// TwinCAT 3 PLC project WashingMachineSimulator
// ProgramVersion: 3.1.4024.0
// libraries:
//   Tc2_Standard, * (Beckhoff Automation GmbH)
//   Tc2_System, * (Beckhoff Automation GmbH)
//   Tc3_Module, * (Beckhoff Automation GmbH)
// project tree:
//   / Class Diagram.TcCD (not stored), PlcTask.TcTTO
//   DUTs/ E_MachineState.TcDUT, E_Strategy.TcDUT, ST_Wash.TcDUT
//   GVLs/ GVL_References.TcGVL
//   POUs/ Class Diagram_1.TcCD (not stored), Class Diagram_2.TcCD (not stored), FB_WashingMachine.TcPOU, MAIN.TcPOU
//   POUs/Motor/ FB_BaseMotor.TcPOU, I_Motor.TcIO
//   POUs/Pump/ FB_WaterController.TcPOU, I_WaterController.TcIO
//   POUs/Strategies/ FB_HeavyWash.TcPOU, FB_NormalWash.TcPOU, FB_SoftWash.TcPOU, I_WashStrategy.TcIO
// real-time tasks:
//   TASK PlcTask: cycle T#10ms, priority 20, ADS port 350

CONFIGURATION WashingMachineSimulator
    RESOURCE PLC ON TwinCAT3
        TASK PlcTask(INTERVAL := T#10ms, PRIORITY := 20);
        PROGRAM MAIN WITH PlcTask : MAIN;
    END_RESOURCE
END_CONFIGURATION

// ---- DUTs/E_MachineState.TcDUT
{attribute 'qualified_only'}
{attribute 'strict'}
TYPE E_MachineState :
(
	IDLE := 0,
	CONFIGURING,
	FILLING,
	WASHING,
	DRAINING,
	COMPLETED,
	DRYING,
	ERROR
);
END_TYPE

// ---- DUTs/E_Strategy.TcDUT
{attribute 'qualified_only'}
{attribute 'strict'}
TYPE E_Strategy :
(
	SOFT := 0,
	NORMAL,
	HEAVY
);
END_TYPE

// ---- DUTs/ST_Wash.TcDUT
TYPE ST_Wash :
STRUCT
	nWaterLevel : INT := 1 ;
	eWashStrategy : E_Strategy := E_Strategy.SOFT;
	
END_STRUCT
END_TYPE

// ---- GVLs/GVL_References.TcGVL
{attribute 'qualified_only'}
VAR_GLOBAL
	fbSoftWash : FB_SoftWash;
	fbNormalWash : FB_NormalWash;
	fbHeavyWash : FB_HeavyWash;
	
	fbMotor : FB_BaseMotor;
	fbWaterController : FB_WaterController;
END_VAR

// ---- POUs/Motor/I_Motor.TcIO
INTERFACE I_Motor

METHOD DrySpin 
VAR_INPUT
	nMotorSpeed : INT;
END_VAR
END_METHOD

METHOD Stop
VAR_INPUT
END_VAR
END_METHOD

METHOD WashSpin 
VAR_INPUT
	nMotorSpeed : INT;
END_VAR
END_METHOD

END_INTERFACE

// ---- POUs/Pump/I_WaterController.TcIO
INTERFACE I_WaterController

METHOD GetDuration : TIME
VAR_INPUT
	stWash : REFERENCE TO ST_Wash;
END_VAR
END_METHOD

METHOD StartDrain : BOOL
VAR_INPUT
END_VAR
END_METHOD

METHOD StartFill : BOOL
VAR_INPUT
END_VAR
END_METHOD

METHOD Stop
END_METHOD

END_INTERFACE

// ---- POUs/Strategies/I_WashStrategy.TcIO
INTERFACE I_WashStrategy

METHOD GetDuration : TIME
END_METHOD

METHOD GetRinseCount : INT
END_METHOD

METHOD StartSpin : BOOL
END_METHOD

METHOD StartWash : BOOL
VAR_INPUT
	iMotor : I_Motor;
END_VAR
END_METHOD

METHOD Stop
END_METHOD

END_INTERFACE

// ---- POUs/MAIN.TcPOU
PROGRAM MAIN
VAR
	stWash1 : ST_Wash := (nWaterLevel := 4, eWashStrategy := E_Strategy.NORMAL );
	
	fbWashingMachine : FB_WashingMachine();
	bStart: BOOL;
	
	eWashingMachineState : E_MachineState;
	tRemainingTime : TIME;
END_VAR

IF bStart THEN
	fbWashingMachine.Start();
END_IF
fbWashingMachine(stWash := stWash1);
eWashingMachineState := fbWashingMachine.eState;
tRemainingTime := fbWashingMachine.tRemainingTime;

END_PROGRAM

// ---- POUs/FB_WashingMachine.TcPOU
FUNCTION_BLOCK FB_WashingMachine

VAR_IN_OUT
	stWash : ST_Wash;
END_VAR
VAR
	iWashStrategy : I_WashStrategy;
	iMotor : I_Motor;
	iWaterController : I_WaterController;
	
	eMachineState : E_MachineState;
	tTotalTime : TIME ;
	bRunning : BOOL;
	tBaseTime : TIME := T#5S;
	tRemainingWashingTime : TIME ;
	nRinseCount : INT;
	
	fbTimer : TON ;
END_VAR


IF tTotalTime <> T#0S THEN
	fbTimer (IN := bRunning , PT := tTotalTime);
	tRemainingTime := fbTimer.PT - fbTimer.ET;
END_IF

IF __ISVALIDREF(stWash) THEN
	
	CASE eMachineState OF
		E_MachineState.IDLE:
			IF bRunning THEN
				eMachineState := E_MachineState.CONFIGURING;
			END_IF
			
		E_MachineState.CONFIGURING:
			nRinseCount := 0;
			iWashStrategy := SelectStrategy();
			iMotor := SelectMotor();
			iWaterController := SelectWaterController();
			IF iWashStrategy <> 0 AND iWaterController <> 0 AND iMotor <> 0 THEN
				tTotalTime := iWaterController.GetDuration(stWash) * iWashStrategy.GetRinseCount() + iWashStrategy.GetDuration();
				tRemainingTime := tTotalTime;
				eMachineState := E_MachineState.FILLING;
			ELSE
				eMachineState := E_MachineState.ERROR;
			END_IF
		
		E_MachineState.FILLING:
			IF NOT iWaterController.StartFill() THEN
				eMachineState := E_MachineState.WASHING;
			END_IF
				
		E_MachineState.WASHING:
			IF iWashStrategy.StartWash(iMotor) THEN
				eMachineState := E_MachineState.DRAINING;
			END_IF
		
		E_MachineState.DRAINING:
				IF NOT iWaterController.StartDrain() THEN
					nRinseCount := nRinseCount + 1;
					IF nRinseCount = iWashStrategy.GetRinseCount() THEN
						eMachineState := E_MachineState.DRYING;
					ELSE
						eMachineState := E_MachineState.FILLING;
					END_IF
				END_IF
				
		E_MachineState.DRYING:
			IF iWashStrategy.StartSpin() THEN
				eMachineState := E_MachineState.COMPLETED;
			END_IF
			
		E_MachineState.COMPLETED:
			Stop();
			fbTimer( IN := bRunning);
			tTotalTime := T#0S;
			tRemainingTime := tTotalTime;
			
		E_MachineState.ERROR:
			Stop();
			
		
	END_CASE
	
END_IF

PROPERTY eState : E_MachineState
GET
eState := eMachineState;
END_GET
SET // PRIVATE
eMachineState := eState;
END_SET
END_PROPERTY

METHOD PRIVATE SelectMotor : I_Motor
SelectMotor := GVL_References.fbMotor;
END_METHOD

METHOD PRIVATE SelectStrategy : I_WashStrategy
CASE stWash.eWashStrategy OF
	E_Strategy.SOFT :
	SelectStrategy :=  GVL_References.fbSoftWash;
	
	E_Strategy.NORMAL :
	SelectStrategy :=  GVL_References.fbNormalWash;
	
	E_Strategy.HEAVY :
	SelectStrategy :=  GVL_References.fbHeavyWash;
	
END_CASE
END_METHOD

METHOD PRIVATE SelectWaterController : I_WaterController
SelectWaterController :=  GVL_References.fbWaterController;
END_METHOD

METHOD Start
bRunning := TRUE;
END_METHOD

METHOD Stop
bRunning := FALSE;
END_METHOD

PROPERTY tRemainingTime : TIME
GET
tRemainingTime := tRemainingWashingTime;
END_GET
SET // PRIVATE
tRemainingWashingTime := tRemainingTime;
END_SET
END_PROPERTY

END_FUNCTION_BLOCK

// ---- POUs/Strategies/FB_SoftWash.TcPOU
FUNCTION_BLOCK FB_SoftWash IMPLEMENTS I_WashStrategy

VAR
	nWashCount : INT := 1;
	nRinseCount : INT := 1;
	iMotorRef : I_Motor;
	bWashing : BOOL;
	bDrying : BOOL;
	
	tWashTime : TIME := T#10S;
	nMotorWashSpeed : INT := 100;
	
	nMotorDrySpeed : INT := 700; 
	nMotorDryTime : TIME := T#7S;
	
	fbWashTimer : TON;
END_VAR

{warning 'add method implementation '}
METHOD GetDuration : TIME
VAR
END_VAR
GetDuration := tWashTime * (nRinseCount + nWashCount) + nMotorDryTime ;
END_METHOD

METHOD GetRinseCount : INT
VAR_INPUT
END_VAR
GetRinseCount := nRinseCount + nWashCount;
END_METHOD

METHOD StartSpin : BOOL
bDrying := TRUE;
fbWashTimer( IN := bDrying, PT := nMotorDryTime);
IF NOT fbWashTimer.Q THEN
	iMotorRef.DrySpin(nMotorDrySpeed);
ELSE
	iMotorRef.Stop();
	bDrying := FALSE;
	fbWashTimer( IN := bDrying);
	StartSpin := TRUE;
END_IF
END_METHOD

{warning 'add method implementation '}
METHOD StartWash : BOOL
VAR_INPUT
	iMotor : I_Motor;
END_VAR
iMotorRef := iMotor;
bWashing := TRUE;
fbWashTimer( IN := bWashing, PT := tWashTime);
IF NOT fbWashTimer.Q THEN
	iMotorRef.WashSpin(nMotorWashSpeed);
ELSE
	iMotorRef.Stop();
	bWashing := FALSE;
	fbWashTimer( IN := bWashing);
	StartWash := TRUE;
END_IF
END_METHOD

{warning 'add method implementation '}
METHOD Stop
bWashing := FALSE;
END_METHOD

END_FUNCTION_BLOCK

// ---- POUs/Strategies/FB_NormalWash.TcPOU
FUNCTION_BLOCK FB_NormalWash IMPLEMENTS I_WashStrategy
VAR
	nWashCount : INT := 1;
	nRinseCount : INT := 2;
	iMotorRef : I_Motor;
	bWashing : BOOL;
	bDrying : BOOL;
	
	tWashTime : TIME := T#15S;
	nMotorWashSpeed : INT := 200;
	
	nMotorDrySpeed : INT := 850; 
	nMotorDryTime : TIME := T#10S;
	
	fbWashTimer : TON;
END_VAR

{warning 'add method implementation '}
METHOD GetDuration : TIME
VAR
END_VAR
GetDuration := tWashTime * (nRinseCount + nWashCount) + nMotorDryTime ;
END_METHOD

METHOD GetRinseCount : INT
VAR_INPUT
END_VAR
GetRinseCount := nRinseCount + nWashCount;
END_METHOD

METHOD StartSpin : BOOL
VAR_INPUT
END_VAR
bDrying := TRUE;
fbWashTimer( IN := bDrying, PT := nMotorDryTime);
IF NOT fbWashTimer.Q THEN
	iMotorRef.DrySpin(nMotorDrySpeed);
ELSE
	iMotorRef.Stop();
	bDrying := FALSE;
	fbWashTimer( IN := bDrying);
	StartSpin := TRUE;
END_IF
END_METHOD

{warning 'add method implementation '}
METHOD StartWash : BOOL
VAR_INPUT
	iMotor : I_Motor;
END_VAR
iMotorRef := iMotor;
bWashing := TRUE;
fbWashTimer( IN := bWashing, PT := tWashTime);
IF NOT fbWashTimer.Q THEN
	iMotorRef.WashSpin(nMotorWashSpeed);
ELSE
	iMotorRef.Stop();
	bWashing := FALSE;
	fbWashTimer( IN := bWashing);
	StartWash := TRUE;
END_IF
END_METHOD

{warning 'add method implementation '}
METHOD Stop
bWashing := FALSE;
END_METHOD

END_FUNCTION_BLOCK

// ---- POUs/Strategies/FB_HeavyWash.TcPOU
FUNCTION_BLOCK FB_HeavyWash IMPLEMENTS I_WashStrategy
VAR
	nWashCount : INT := 1;
	nRinseCount : INT := 3;
	iMotorRef : I_Motor;
	bWashing : BOOL;
	bDrying : BOOL;
	
	tWashTime : TIME := T#20S;
	nMotorWashSpeed : INT := 300;
	
	nMotorDrySpeed : INT := 1000; 
	nMotorDryTime : TIME := T#15S;
	
	fbWashTimer : TON;
END_VAR

{warning 'add method implementation '}
METHOD GetDuration : TIME
VAR
END_VAR
GetDuration := tWashTime * (nRinseCount + nWashCount) + nMotorDryTime ;
END_METHOD

METHOD GetRinseCount : INT
VAR_INPUT
END_VAR
GetRinseCount := nRinseCount + nWashCount;
END_METHOD

METHOD StartSpin : BOOL
VAR_INPUT
END_VAR
bDrying := TRUE;
fbWashTimer( IN := bDrying, PT := nMotorDryTime);
IF NOT fbWashTimer.Q THEN
	iMotorRef.DrySpin(nMotorDrySpeed);
ELSE
	iMotorRef.Stop();
	bDrying := FALSE;
	fbWashTimer( IN := bDrying);
	StartSpin := TRUE;
END_IF
END_METHOD

{warning 'add method implementation '}
METHOD StartWash : BOOL
VAR_INPUT
	iMotor : I_Motor;
END_VAR
iMotorRef := iMotor;
bWashing := TRUE;
fbWashTimer( IN := bWashing, PT := tWashTime);
IF NOT fbWashTimer.Q THEN
	iMotorRef.WashSpin(nMotorWashSpeed);
ELSE
	iMotorRef.Stop();
	bWashing := FALSE;
	fbWashTimer( IN := bWashing);
	StartWash := TRUE;
END_IF
END_METHOD

{warning 'add method implementation '}
METHOD Stop
bWashing := FALSE;
END_METHOD

END_FUNCTION_BLOCK

// ---- POUs/Motor/FB_BaseMotor.TcPOU
FUNCTION_BLOCK FB_BaseMotor IMPLEMENTS I_Motor

VAR
	nMotorSpeed : INT;
	bEnable : BOOL;
END_VAR

{warning 'add method implementation '}
METHOD DrySpin
VAR_INPUT
	nMotorSpeed	: INT;
END_VAR
bEnable := TRUE;
This^.nMotorSpeed := nMotorSpeed;
END_METHOD

METHOD Stop
bEnable := FALSE;
END_METHOD

{warning 'add method implementation '}
METHOD WashSpin
VAR_INPUT
	nMotorSpeed	: INT;
END_VAR
bEnable := TRUE;
This^.nMotorSpeed := nMotorSpeed;
END_METHOD

END_FUNCTION_BLOCK

// ---- POUs/Pump/FB_WaterController.TcPOU
FUNCTION_BLOCK FB_WaterController IMPLEMENTS I_WaterController

VAR
	bInletValve : BOOL;
	bOutletValve : BOOL;
	
	tBaseTime : TIME := T#5S;
	tFillingTime : TIME ;
	tDrainingTime : TIME ;
	
	fbWaterTimer : TON;
END_VAR

METHOD GetDuration : TIME
VAR_INPUT
	stWash : REFERENCE TO ST_Wash;
END_VAR

tFillingTime := tBaseTime * stWash.nWaterLevel;
tDrainingTime := tBaseTime * stWash.nWaterLevel;
GetDuration := tFillingTime + tDrainingTime;
END_METHOD

{warning 'add method implementation '}
METHOD StartDrain : BOOL

StartDrain := bOutletValve := TRUE;
fbWaterTimer( IN := bOutletValve, PT := tFillingTime);
IF fbWaterTimer.Q THEN
	bOutletValve := FALSE;
	StartDrain := FALSE;
	fbWaterTimer( IN := bOutletValve);
END_IF
END_METHOD

{warning 'add method implementation '}
METHOD StartFill : BOOL
StartFill := bInletValve := TRUE;
fbWaterTimer( IN := bInletValve, PT := tFillingTime);
IF fbWaterTimer.Q THEN
	bInletValve := FALSE;
	StartFill := FALSE;
	fbWaterTimer( IN := bInletValve);
END_IF
END_METHOD

METHOD Stop
bInletValve := bOutletValve := FALSE;
END_METHOD

END_FUNCTION_BLOCK
